Yaskawa INFORM job: TEST_R2.JBI

/JOB
//NAME TEST_R2
///FOLDERNAME INNE
//POS
///NPOS 4,4,0,0,0,0
///TOOL 0
///POSTYPE PULSE
///PULSE
C00000=79854,52857,64617,69830,29819,-35293
C00001=117495,-36235,-69384,1898,67215,-1067
C00002=79745,53967,65773,70095,29839,-35439
C00003=118404,41237,-3817,1368,66658,-772
BC00000=398161,156221,441640
BC00001=14348,232885,967813
BC00002=398161,1155144,441640
BC00003=14348,1312767,967813
//INST
///DATE 2023/11/01 18:40
///ATTR SC,RW
///GROUP1 RB1,BS1
NOP
'test_R2
MOVJ C00000 BC00000 VJ=100.00
MOVJ C00001 BC00001 VJ=100.00
MOVJ C00002 BC00002 VJ=100.00
MOVJ C00003 BC00003 VJ=100.00
END
